SYSTEM MVCTest (* System Configuration *)
  (* Standard: 61499-1 *)
  (* Version 0.3, 2003-12-05, JHC, Rockwell Automation, Renamed from NEWSYSTEM. *)
  (* Version 0.2, 2002-11-05, JHC, Rockwell Automation, Fixed missing (empty) FBD in Application. *)
  (* Version 0.1, 2002-01-17, JHC, Rockwell Automation, Minor cleanup *)
  (* Version 0.0, 2000-05-27, JHC, Rockwell Automation *)
  APPLICATION APP1
  END_APPLICATION
  DEVICE HMI : FRAME_DEVICE(BOUNDS := [10,10,100,200], GRID := [2,1])
    RESOURCE Test : PANEL_RESOURCE
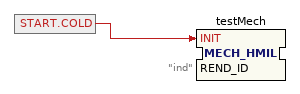
      FBS
        testMech : MECH_HMIL(REND_ID := "ind");
      END_FBS
      EVENT_CONNECTIONS
        START.COLD TO testMech.INIT;
      END_CONNECTIONS
    END_RESOURCE
    RESOURCE RES1 : PANEL_RESOURCE
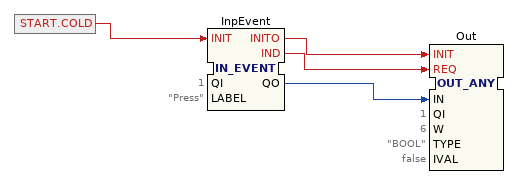
      FBS
        InpEvent : IN_EVENT(QI := 1, LABEL := "Press");
        Out : OUT_ANY(QI := 1, W := 6, TYPE := "BOOL", IVAL := false);
      END_FBS
      EVENT_CONNECTIONS
        START.COLD TO InpEvent.INIT;
        InpEvent.INITO TO Out.INIT;
        InpEvent.IND TO Out.REQ;
      END_CONNECTIONS
      DATA_CONNECTIONS
        InpEvent.QO TO Out.IN;
      END_CONNECTIONS
    END_RESOURCE
  END_DEVICE
  DEVICE View : FRAME_DEVICE(BOUNDS := [10,210,200,200])
    RESOURCE ViewPanel : PANEL_RESOURCE
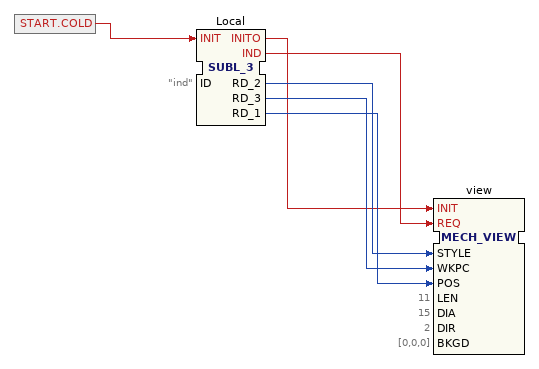
      FBS
        view : MECH_VIEW(LEN := 11, DIA := 15, DIR := 2, BKGD := [0,0,0]);
        Local : SUBL_3(ID := "ind");
      END_FBS
      EVENT_CONNECTIONS
        START.COLD TO Local.INIT;
        Local.INITO TO view.INIT;
        Local.IND TO view.REQ;
      END_CONNECTIONS
      DATA_CONNECTIONS
        Local.RD_2 TO view.STYLE;
        Local.RD_3 TO view.WKPC;
        Local.RD_1 TO view.POS;
      END_CONNECTIONS
    END_RESOURCE
  END_DEVICE
END_SYSTEM
